PROGRAM PRG_SP1K2_PAX
VAR
	bInit : BOOL := TRUE;
	fbPAX_TAR_X : FB_MotionStage;
	fbPAX_TAR_Y : FB_MotionStage;
	fbPAX_TAR_Z : FB_MotionStage;
	
	fbPAX_BB_Y_01 : FB_MotionStage;
	fbPAX_BB_Y_02 : FB_MotionStage;
END_VAR

IF bInit THEN
	Main.M28.bHardwareEnable := TRUE;
	Main.M29.bHardwareEnable := TRUE;
	Main.M30.bHardwareEnable := TRUE;
	Main.M31.bHardwareEnable := TRUE;
	Main.M32.bHardwareEnable := TRUE;
	Main.M33.bHardwareEnable := TRUE;
	Main.M34.bHardwareEnable := TRUE;
	bInit := FALSE;
END_IF

fbPAX_TAR_X(stMotionStage:= Main.M32);
fbPAX_TAR_Y(stMotionStage:= Main.M33);
fbPAX_TAR_Z(stMotionStage:= Main.M34);

fbPAX_BB_Y_01(stMotionStage:= Main.M36);
fbPAX_BB_Y_02(stMotionStage:= Main.M37);

END_PROGRAM

(* stored: Version 1.1.0.1, ProductVersion 3.1.4022.18
   POU PRG_SP1K2_PAX: Id {7594ee7f-4f5d-4eba-b4fd-40f8476ab083}, SpecialFunc None *)
